TYPE ST_Array :
STRUCT
	IntArr  : ARRAY [0..8] OF INT	  ;
	RealArr  : ARRAY [0..25] OF REAL	  ;
	BoolArr  : ARRAY [0..25] OF BOOL	  ;

END_STRUCT
END_TYPE

(* stored: Version 1.1.0.1, ProductVersion 3.1.4024.12
   DUT ST_Array: Id {4fd8cd4a-bb46-407b-8461-1eb3a60a02ce} *)
